// TIA Portal project "2022.06.08_FB参数" (V17)

(* hardware
DEVICE "S7-1200 station_1"  S7-1200 Station
   slot 0: "Rack_0"  S7-1200 Rack  Rack  V1.0
   slot 1: "PLC_1"  CPU 1212C DC/DC/DC  6ES7 212-1AE40-0XB0  V4.5
*)

// ===== PLC "PLC_1"  CPU 1212C DC/DC/DC =====

VAR_GLOBAL   // PLC tag table "默认变量表"
   "模拟量输入" AT %MW100 : Word;
   "Tag_3" AT %MW102 : UInt;
   "Tag_4" AT %MW104 : UInt;
   "Tag_5" AT %MW106 : UInt;
   "Tag_6" AT %I0.0 : Bool;
   "Tag_7" AT %M0.0 : Bool;
   "X(2)" AT %MW10 : Word;
   "Tag_9" AT %MW12 : UInt;
   "X" AT %MW0 : Word;
   "a" AT %MW2 : Word;
   "b" AT %MW4 : Int;
   "c" AT %MW8 : Int;
   "实时温度" AT %MD0 : Real;
   "Tag_10" AT %MD2 : Real;
   "f" AT %MD4 : Real;
   "g" AT %MD8 : Real;
   "X(1)" AT %MD12 : Real;
   "Tag_8" AT %MD16 : Real;
   "中间值(1)" AT %MD200 : Real;
   "中间值" AT %MD104 : Real;
   "工程值" AT %MD108 : Real;
   "要求的频率" AT %MD60 : Real;
   "百分比" AT %MD64 : Real;
   "Tag_12" AT %MW70 : Int;
   "Tag_2" AT %I0.1 : Bool;
   "0" AT %Q0.0 : Bool;
   "加热" AT %Q0.1 : Bool;
   "Tag_1" AT %MD100 : Time;
   "Tag_11" AT %M0.1 : Bool;
   "Tag_13" AT %QB0 : Byte;
   "Tag_14" AT %QB1 : Byte;
   "Tag_15" AT %M0.2 : Bool;
   "Tag_16" AT %QB2 : Byte;
   "Tag_17" AT %I0.2 : Bool;
   "Tag_18" AT %M10.0 : Bool;
   "Tag_19" AT %Q0.2 : Bool;
   "Tag_20" AT %I0.3 : Bool;
   "Tag_21" AT %I0.4 : Bool;
   "Tag_22" AT %Q0.3 : Bool;
   "Tag_23" AT %Q0.4 : Bool;
   "Tag_24" AT %Q0.5 : Bool;
   "Tag_25" AT %MD6 : Real;
END_VAR

DATA_BLOCK "一元二次方程_DB"   // DB1
{ S7_Optimized_Access := 'TRUE' }
VERSION : 0.1
// stored: InstanceOfName 一元二次方程
"一元二次方程"
BEGIN
END_DATA_BLOCK

FUNCTION_BLOCK "一元二次方程"   // FB1, LAD
{ S7_Optimized_Access := 'TRUE' }
VERSION : 0.1
   VAR_INPUT
      x : Real;
   END_VAR
   VAR_OUTPUT
      y : Real;
   END_VAR
   VAR
      "a" : Real;
      "b" : Real;
      c : Real;
   END_VAR
BEGIN

REGION Network 1
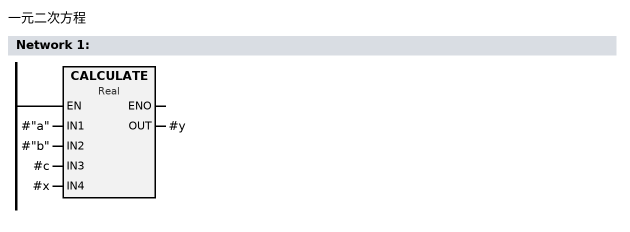
   RUNG wire#powerrail
      { S7_Templates := "SrcType := Real"; S7_Expression := "IN1*SQRT(IN4)+IN2*IN4+IN3" } Calculate(in1 := #"a", in2 := #"b", in3 := #c, in4 := #x, out => #y)
   END_RUNG
   // the same network as SCL:
   #y := #"a"*SQRT(#x)+#"b"*#x+#c;
END_REGION
END_FUNCTION_BLOCK

ORGANIZATION_BLOCK "Main"   // OB1, LAD, ProgramCycle
TITLE = "Main Program Sweep (Cycle)"
{ S7_Optimized_Access := 'TRUE' }
VERSION : 0.1
   VAR_INPUT
      Initial_Call : Bool;   // Initial call of this OB
      Remanence : Bool;   // =True, if remanent data are available
   END_VAR
BEGIN

REGION Network 1
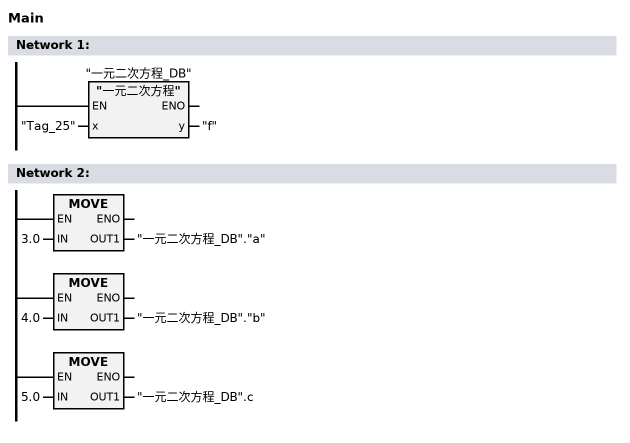
   RUNG wire#powerrail
      "一元二次方程_DB"(x := "Tag_25", y => "f")
   END_RUNG
   // the same network as SCL:
   "一元二次方程_DB"(x := "Tag_25", y => "f");   // "一元二次方程"
END_REGION

REGION Network 2
   RUNG wire#powerrail
      Move(in := 3.0, out1 => "一元二次方程_DB"."a")
   END_RUNG
   RUNG wire#powerrail
      Move(in := 4.0, out1 => "一元二次方程_DB"."b")
   END_RUNG
   RUNG wire#powerrail
      Move(in := 5.0, out1 => "一元二次方程_DB".c)
   END_RUNG
   // the same network as SCL:
   "一元二次方程_DB"."a" := 3.0;
   "一元二次方程_DB"."b" := 4.0;
   "一元二次方程_DB".c := 5.0;
END_REGION
END_ORGANIZATION_BLOCK